FUNCTION_BLOCK CS_DustMoter
VAR_INPUT
END_VAR
VAR_OUTPUT
END_VAR
VAR
END_VAR

VAR_IN_OUT
stSetpMotor:ST_DustMotor;
END_VAR
	

VAR
R_trig20:R_TRIG;
R_trig21:R_TRIG;
F_trig23:F_TRIG;
F_trig22:F_TRIG;
END_VAR

(*********************毛刷步进电机控制*****************************)
//步进点动
stSetpMotor.bo_Pul:=stSetpMotor.bJog_FW OR stSetpMotor.bJog_BW ;   //步进点动正转
stSetpMotor.bo_Dir:=stSetpMotor.bJog_BW ; //步进点动反转   

R_trig20(CLK:=stSetpMotor.bRun_FW , Q=> );
R_trig21(CLK:=stSetpMotor.bRun_BW , Q=> );
F_trig22(CLK:=stSetpMotor.bRun_FW , Q=> );
F_trig23(CLK:=stSetpMotor.bRun_BW , Q=> );
IF R_trig20.Q THEN
   stSetpMotor.bJog_FW:=TRUE;
   stSetpMotor.bJog_BW:=FALSE;
END_IF
IF R_trig21.Q THEN
   stSetpMotor.bJog_FW:=FALSE;
   stSetpMotor.bJog_BW:=TRUE;
END_IF
IF F_trig22.Q OR F_trig23.Q THEN
   stSetpMotor.bJog_FW:=FALSE;
   stSetpMotor.bJog_BW:=FALSE;
END_IF

END_FUNCTION_BLOCK

(* stored: Version 1.1.0.1, ProductVersion 3.1.4024.9
   POU CS_DustMoter: Id {a10c32ae-31b4-4417-ad3e-63486ed7fec2}, SpecialFunc None *)
